PROGRAM prgComEffIO
VAR
	fbCom		: FB_MqttCommunicator_V5;
END_VAR

// CX-7BDACD
fbCom(
	bConnect:= TRUE, 
	strAuthKey := 'ENE87365342998',
	sUserName:= 'a4398363-713f-45e4-8f12-13b95d7f2606', 
	sUserPassword:= '196c948c-aabd-4764-8be4-f15873a2b8fa', 
	eSavePositionCertificate:= eSavePositionOnPLC.ePostionHardDisk,
	time_HeartBeat_sec:= T#50S, 
	bConnected=> , 
	bError=> , 
	hrErrorCode=> , 
	eConnectionState=> , 
	eErrorMessage_Out=> );

END_PROGRAM

(* stored: Version 1.1.0.1, ProductVersion 3.1.4024.13
   POU prgComEffIO: Id {cbcd318b-bf51-484c-bcaa-d6efcdf43fe3}, SpecialFunc None *)
